KUKA KRL program: _Axis_MAIN_dataset.src, _Axis_MAIN_dataset.dat

--- _Axis_MAIN_dataset.src ---
&ACCESS RVP
&REL 8
&PARAM EDITMASK = *
&PARAM TEMPLATE = C:\KRC\Roboter\Template\vorgabe
&PARAM DISKPATH = KRC:\R1\Diagnostika
DEF _Axis_MAIN_dataset ( )
   ;FOLD INI;%{PE}
      ;FOLD BASISTECH INI
         GLOBAL INTERRUPT DECL 3 WHEN $STOPMESS==TRUE DO IR_STOPM ( )
         INTERRUPT ON 3
         BAS (#INITMOV,0 )
      ;ENDFOLD (BASISTECH INI)
      ;FOLD USER INI
         ;Make your modifications here

      ;ENDFOLD (USER INI)
      ;ENDFOLD (INI)
   PyRUN=FALSE
   PyDONE=FALSE
   PySPEED=50
   $ADVANCE = 0
   ;FOLD domu
      SPTP DOMOV WITH $VEL_AXIS[1] = SVEL_JOINT(100), $TOOL = STOOL2(FP1), $BASE = SBASE(FP1.BASE_NO), $IPO_MODE = SIPO_MODE(FP1.IPO_FRAME), $LOAD = SLOAD(FP1.TOOL_NO), $ACC_AXIS[1] = SACC_JOINT(PPDAT1), $APO = SAPO_PTP(PPDAT1), $GEAR_JERK[1] = SGEAR_JERK(PPDAT1), $COLLMON_TOL_PRO[1] = USE_CM_PRO_VALUES(0)
   ;ENDFOLD
   LOOP
      $ANOUT[1]=0
      WAIT FOR PyRUN
      PyDONE = FALSE
      ; $TIMER[1]=0
      $TIMER_STOP[1]=FALSE
      ;FOLD domu
         SPTP DOMOV WITH $VEL_AXIS[1] = SVEL_JOINT(PySPEED), $TOOL = STOOL2(FP1), $BASE = SBASE(FP1.BASE_NO), $IPO_MODE = SIPO_MODE(FP1.IPO_FRAME), $LOAD = SLOAD(FP1.TOOL_NO), $ACC_AXIS[1] = SACC_JOINT(PPDAT1), $APO = SAPO_PTP(PPDAT1), $GEAR_JERK[1] = SGEAR_JERK(PPDAT1), $COLLMON_TOL_PRO[1] = USE_CM_PRO_VALUES(0)
      ;ENDFOLD
      $ANOUT[1]=1
      FOR counter = 0 TO PyITER[1]-1 STEP 1
         A1()
      ENDFOR
      $ANOUT[1]=0
      ;FOLD domu
         SPTP DOMOV WITH $VEL_AXIS[1] = SVEL_JOINT(PySPEED), $TOOL = STOOL2(FP1), $BASE = SBASE(FP1.BASE_NO), $IPO_MODE = SIPO_MODE(FP1.IPO_FRAME), $LOAD = SLOAD(FP1.TOOL_NO), $ACC_AXIS[1] = SACC_JOINT(PPDAT1), $APO = SAPO_PTP(PPDAT1), $GEAR_JERK[1] = SGEAR_JERK(PPDAT1), $COLLMON_TOL_PRO[1] = USE_CM_PRO_VALUES(0)
      ;ENDFOLD
      $ANOUT[1]=2
      FOR counter = 0 TO PyITER[2]-1 STEP 1
         A2()
      ENDFOR
      $ANOUT[1]=0
      ;FOLD domu
         SPTP DOMOV WITH $VEL_AXIS[1] = SVEL_JOINT(PySPEED), $TOOL = STOOL2(FP1), $BASE = SBASE(FP1.BASE_NO), $IPO_MODE = SIPO_MODE(FP1.IPO_FRAME), $LOAD = SLOAD(FP1.TOOL_NO), $ACC_AXIS[1] = SACC_JOINT(PPDAT1), $APO = SAPO_PTP(PPDAT1), $GEAR_JERK[1] = SGEAR_JERK(PPDAT1), $COLLMON_TOL_PRO[1] = USE_CM_PRO_VALUES(0)
      ;ENDFOLD
      $ANOUT[1]=3
      FOR counter = 0 TO PyITER[3]-1 STEP 1
         A3()
      ENDFOR
      $ANOUT[1]=0
      ;FOLD domu
         SPTP DOMOV WITH $VEL_AXIS[1] = SVEL_JOINT(PySPEED), $TOOL = STOOL2(FP1), $BASE = SBASE(FP1.BASE_NO), $IPO_MODE = SIPO_MODE(FP1.IPO_FRAME), $LOAD = SLOAD(FP1.TOOL_NO), $ACC_AXIS[1] = SACC_JOINT(PPDAT1), $APO = SAPO_PTP(PPDAT1), $GEAR_JERK[1] = SGEAR_JERK(PPDAT1), $COLLMON_TOL_PRO[1] = USE_CM_PRO_VALUES(0)
      ;ENDFOLD
      $ANOUT[1]=4
      FOR counter = 0 TO PyITER[4]-1 STEP 1
         A4()
      ENDFOR
      $ANOUT[1]=0
      ;FOLD domu
         SPTP DOMOV WITH $VEL_AXIS[1] = SVEL_JOINT(PySPEED), $TOOL = STOOL2(FP1), $BASE = SBASE(FP1.BASE_NO), $IPO_MODE = SIPO_MODE(FP1.IPO_FRAME), $LOAD = SLOAD(FP1.TOOL_NO), $ACC_AXIS[1] = SACC_JOINT(PPDAT1), $APO = SAPO_PTP(PPDAT1), $GEAR_JERK[1] = SGEAR_JERK(PPDAT1), $COLLMON_TOL_PRO[1] = USE_CM_PRO_VALUES(0)
      ;ENDFOLD
      $ANOUT[1]=5
      FOR counter = 0 TO PyITER[5]-1 STEP 1
         A5()
      ENDFOR
      $ANOUT[1]=0
      ;FOLD domu
         SPTP DOMOV WITH $VEL_AXIS[1] = SVEL_JOINT(PySPEED), $TOOL = STOOL2(FP1), $BASE = SBASE(FP1.BASE_NO), $IPO_MODE = SIPO_MODE(FP1.IPO_FRAME), $LOAD = SLOAD(FP1.TOOL_NO), $ACC_AXIS[1] = SACC_JOINT(PPDAT1), $APO = SAPO_PTP(PPDAT1), $GEAR_JERK[1] = SGEAR_JERK(PPDAT1), $COLLMON_TOL_PRO[1] = USE_CM_PRO_VALUES(0)
      ;ENDFOLD
      $ANOUT[1]=6
      FOR counter = 0 TO PyITER[6]-1 STEP 1
         A6()
      ENDFOR
      $ANOUT[1]=0
      ;FOLD domu
         SPTP DOMOV WITH $VEL_AXIS[1] = SVEL_JOINT(PySPEED), $TOOL = STOOL2(FP1), $BASE = SBASE(FP1.BASE_NO), $IPO_MODE = SIPO_MODE(FP1.IPO_FRAME), $LOAD = SLOAD(FP1.TOOL_NO), $ACC_AXIS[1] = SACC_JOINT(PPDAT1), $APO = SAPO_PTP(PPDAT1), $GEAR_JERK[1] = SGEAR_JERK(PPDAT1), $COLLMON_TOL_PRO[1] = USE_CM_PRO_VALUES(0)
      ;ENDFOLD
      WAIT SEC 0
      PyDONE = TRUE
      PyRUN = FALSE
      ColRUN = FALSE
      $TIMER_STOP[1]=TRUE
      WAIT SEC 1
      PyDONE = FALSE
   ENDLOOP
END

--- _Axis_MAIN_dataset.dat ---
&ACCESS RVP
&REL 8
&PARAM EDITMASK = *
&PARAM TEMPLATE = C:\KRC\Roboter\Template\vorgabe
&PARAM DISKPATH = KRC:\R1\Diagnostika
DEFDAT  _Axis_MAIN_dataset
;FOLD EXTERNAL DECLARATIONS;%{PE}%MKUKATPBASIS,%CEXT,%VCOMMON,%P
;FOLD BASISTECH EXT;%{PE}%MKUKATPBASIS,%CEXT,%VEXT,%P
EXT  BAS (BAS_COMMAND  :IN,REAL  :IN )

;ENDFOLD (BASISTECH EXT)
;FOLD USER EXT;%{E}%MKUKATPUSER,%CEXT,%VEXT,%P
;Make your modifications here
DECL INT counter
DECL AXIS DOMOV={A1 0.0,A2 -90.0000,A3 90.0000,A4 0.0,A5 60.0000,A6 0.0}
DECL FDAT FP1={TOOL_NO 1,BASE_NO 0,IPO_FRAME #BASE,POINT2[] " "}
DECL PDAT PPDAT1={VEL 100.000,ACC 100.000,APO_DIST 500.000,APO_MODE #CDIS,GEAR_JERK 100.000,EXAX_IGN 0}
;ENDFOLD (USER EXT)
;ENDFOLD (EXTERNAL DECLARATIONS)

ENDDAT
